(* PLC project master, Dassault Systèmes ControlBuild 2024x *)
(* stored: creationDateTime 2023-10-03T11:13:40-01:00 *)

FUNCTION_BLOCK bottling_line.master
  VAR_INPUT
    startCyclePB : BOOL := false;
    initPB : BOOL := false;
    preparationPB : BOOL := false;
    productionPB : BOOL := false;
    closingPB : BOOL := false;
  END_VAR
  VAR_INPUT
    initEnd : BOOL := false;
    preparationEnd : BOOL := false;
    closingEnd : BOOL := false;
    lowLevel3 : BOOL := false;
  END_VAR
  VAR_OUTPUT
    initializationRqst : BOOL := false;
    preparationRqst : BOOL := false;
    productionRqst : BOOL := false;
    closingRqst : BOOL := false;
  END_VAR
  VAR_OUTPUT
    masterInStandBy : BOOL := false;
    productionWaiting : BOOL := false;
  END_VAR

INITIAL_STEP 10:
  10_INLINE1(N);
  COMPUTE_FUNCTION_BLOCKS(S);
END_STEP
ACTION 10_INLINE1:
  masterInStandBy;
END_ACTION
TRANSITION FROM 10 TO 11
  := startCyclePB;
END_TRANSITION
STEP 11:
END_STEP
TRANSITION FROM 11 TO 12
  := initPB;
END_TRANSITION
TRANSITION FROM 11 TO 13
  := preparationPB;
END_TRANSITION
TRANSITION FROM 11 TO 16
  := closingPB;
END_TRANSITION
STEP 12:
  12_INLINE2(N);
END_STEP
ACTION 12_INLINE2:
  initializationRqst;
END_ACTION
TRANSITION FROM 12 TO 10
  := initEnd;
END_TRANSITION
STEP 13:
  13_INLINE3(N);
END_STEP
ACTION 13_INLINE3:
  preparationRqst;
END_ACTION
TRANSITION FROM 13 TO 14
  := preparationEnd;
END_TRANSITION
STEP 16:
  16_INLINE4(N);
END_STEP
ACTION 16_INLINE4:
  closingRqst;
END_ACTION
TRANSITION FROM 16 TO 10
  := closingEnd;
END_TRANSITION
STEP 14:
  14_INLINE5(N);
END_STEP
ACTION 14_INLINE5:
  productionWaiting;
END_ACTION
TRANSITION FROM 14 TO 15
  := productionPB;
END_TRANSITION
STEP 15:
  15_INLINE6(N);
END_STEP
ACTION 15_INLINE6:
  productionRqst;
END_ACTION
TRANSITION FROM 15 TO 13
  := lowLevel3;
END_TRANSITION
TRANSITION FROM 15 TO 10
  := NOT productionPB;
END_TRANSITION
ACTION COMPUTE_FUNCTION_BLOCKS:  (* blocks drawn on the SFC sheet *)
  G1:
END_ACTION
END_FUNCTION_BLOCK
